Fanuc KAREL source: kt00020.KL

-- PROVISIONAL review KL for V1013-1; original PC SHA256 a0379185084ad9c35eda1898d5907ce90b8a8ec4aa0e4c4ea6c19584ec24f06f
-- Incomplete behavior may be omitted. Consult companion uncertainty JSON. Do not deploy.
PROGRAM KT00020
%NOLOCKGROUP
VAR
  R2 : REAL
  OUT : REAL
-- UNRESOLVED_DECL Y1 type=002018
BEGIN
  -- UNRESOLVED_PC offsets 5-19; opcodes 2E,22,9D,33,B2
  -- UNRESOLVED_PC offsets 24-35; opcodes 2E,23
  -- UNRESOLVED_PC offsets 40-64; opcodes 22,9D,33,B1,21,29,64,69,23
  -- UNRESOLVED_PC offsets 69-73; opcodes 7F
END KT00020
